% RSLogix 500 project MOTOR FORWARD & REVERSE INTERLOCK PROTECTION_BAK012.RSS, saved by version 8.30.00.16 %
PROJECT "UNTITLED"    % processor: Bul.1763 MicroLogix 1100 Series B %

PROGRAM FILES
  LAD 2   2 rungs

DATA FILES
  O0 OUTPUT  4 elements
  I1 INPUT  6 elements
  S2 STATUS  66 elements
  B3 BINARY  1 elements
  T4 TIMER  1 elements
  C5 COUNTER  1 elements
  R6 CONTROL  1 elements
  N7 INTEGER  1 elements
  F8 FLOAT  1 elements

LADDER 2
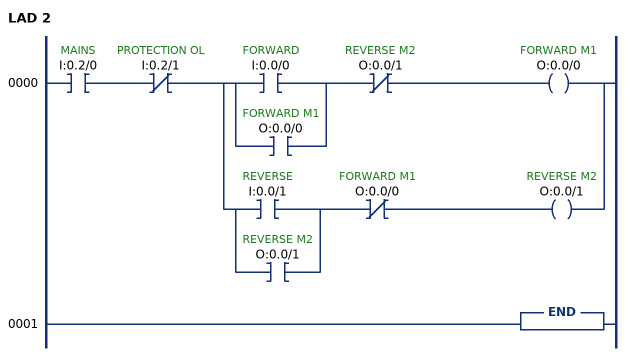
% Rung: 0 %
SOR XIC I:0.2/0 XIO I:0.2/1 BST BST XIC I:0.0/0 NXB XIC O:0.0/0 BND XIO O:0.0/1 OTE O:0.0/0 NXB BST XIC I:0.0/1 NXB XIC O:0.0/1 BND XIO O:0.0/0 OTE O:0.0/1 BND EOR
%   I:0.2/0  MAINS %
%   I:0.2/1  OL  "PROTECTION" %
%   I:0.0/0  FORWARD %
%   O:0.0/0  M1  "FORWARD" %
%   O:0.0/1  M2  "REVERSE" %
%   I:0.0/1  REVERSE %
% Rung: 1 %
SOR END EOR
